(*
Funion block manages the scene data. When rising edge on bSceneON is detected
it recalls a scene from the memory. If rising edge is detected on bSaveScene
it saves the scene to memory under bySceneID number.
Futhermore it save the information about individual lamps being cut off from the scene.
Main idea is that FB uses GVL_IO.arrStreetLamps as 'live buffer' ,
GVL_IO.arrScenes<  > on the other hand is a data 'memory buffer'. 
*)
FUNCTION_BLOCK FB_SceneController
VAR_INPUT
END_VAR
VAR_OUTPUT
	bBusy				:BOOL:=FALSE;		//when TRUE FB is busy working
END_VAR
VAR
	bySceneID			: BYTE;		//number of scene that is being manipulated
	iSelector			: INT := 0;	//variable used in CASE statement
	iCounter			: INT := 0;	//for loop counter
	
	
END_VAR

//if FB is not busy
IF NOT bBusy THEN
	//read BACnet object
	iSelector := REAL_TO_INT(fbBACnet_AV_SL_Scene.fPresentValue);
END_IF

CASE iSelector OF
	0, 255:	//idle state
		;
		
	1..127:	//SceneON
		bBusy := TRUE;	//set a flag indicating that this FB is busy
		
		//reset manual mode
		bBACnet_ResetManual := TRUE;
		
		//convert int to byte
		bySceneID := INT_TO_BYTE(iSelector);
		
		//rewrite power levels from memory buffer to BACnet objects
		fbBACnet_AV_SL_Level_1.fPV  := GVL_IO.arrScenesStreetLampsLevels[bySceneID, 1];
		fbBACnet_AV_SL_Level_2.fPV  := GVL_IO.arrScenesStreetLampsLevels[bySceneID, 2];
		fbBACnet_AV_SL_Level_3.fPV  := GVL_IO.arrScenesStreetLampsLevels[bySceneID, 3];
		fbBACnet_AV_SL_Level_4.fPV  := GVL_IO.arrScenesStreetLampsLevels[bySceneID, 4];
		fbBACnet_AV_SL_Level_5.fPV  := GVL_IO.arrScenesStreetLampsLevels[bySceneID, 5];
		fbBACnet_AV_SL_Level_6.fPV  := GVL_IO.arrScenesStreetLampsLevels[bySceneID, 6];
		fbBACnet_AV_SL_Level_7.fPV  := GVL_IO.arrScenesStreetLampsLevels[bySceneID, 7];
		fbBACnet_AV_SL_Level_8.fPV  := GVL_IO.arrScenesStreetLampsLevels[bySceneID, 8];
		fbBACnet_AV_SL_Level_9.fPV  := GVL_IO.arrScenesStreetLampsLevels[bySceneID, 9];
		fbBACnet_AV_SL_Level_10.fPV := GVL_IO.arrScenesStreetLampsLevels[bySceneID, 10];
			
		iSelector := 0;		//after rewriting data go back to idle
		bBusy := FALSE;		//indicate that this FB is no longer busy
		
		
	128..254:	//SaveScene
		bBusy := TRUE;	//set a flag indicating that this FB is busy
		
		bySceneID := INT_TO_BYTE(iSelector) - 127;
		
		//iterate through arrays to
		FOR iCounter := 1 TO byStreetLampsCount BY 1 DO
			//save current lamp's power levels to memory buffer
			GVL_IO.arrScenesStreetLampsLevels[bySceneID, iCounter]
				:= GVL_IO.arrStreetLamps[iCounter].nLevel;
		END_FOR
		
		iSelector := 0;		//after saving data go back to idle
		bBusy := FALSE;		//indicate that this FB is no longer busy
		
END_CASE

END_FUNCTION_BLOCK

(* stored: Version 1.1.0.1, ProductVersion 3.1.4024.5
   POU FB_SceneController: Id {130ce1fb-8efb-4aa7-9bf7-6373c671b6e1}, SpecialFunc None *)
